// Block: PPrgArchive20

DATA_BLOCK PPrgArchive20
VERSION : 0.1
   NON_RETAIN
   VAR
      PRG : Array[1901..2000] of PPrg_Data;
   END_VAR

BEGIN
   // No initialization required
END_DATA_BLOCK
